PROGRAM CoolingFan
VAR
	bLowFlowTempWarning : BOOL := FALSE;
	bUnloadBoilerToTanks : BOOL := FALSE;
	tonPump2: TON;
END_VAR

// Automatic controll for lauhdutin fan
// Turn fan OFF if in-out temp diff > 10 or out temp < 55 
IF GVL.fTE[15]-GVL.fTE[16] > 10 THEN 
	GVL.bFanPower := FALSE; 
ELSE 
	IF NOT bLowFlowTempWarning THEN
		GVL.bFanPower := TRUE;
	END_IF
END_IF
IF GVL.fTE[15] < 55 THEN // activate low flow temp warning
	bLowFlowTempWarning := TRUE;
	GVL.bFanPower := FALSE;
	GVL.bP3 := FALSE;
	GVL.bHV[11] := FALSE;
END_IF
IF GVl.fTE[15] > 56 THEN
	GVL.bP3 := TRUE;;
	GVL.bHV[11] := TRUE;
END_IF
IF GVL.fTE[15] > 59 THEN  // reset low flow temp warning
	bLowFlowTempWarning := FALSE;
END_IF

END_PROGRAM

(* stored: Version 1.1.0.1, ProductVersion 3.1.4022.18
   POU CoolingFan: Id {f6c82233-30f6-4cd0-a553-a6720ba3592b}, SpecialFunc None *)
